// TIA Portal V20 export
FUNCTION "IF_Bool_Mapping" : Void   // FC104, SCL
// stored: SetENOAutomatically false
BEGIN
       // Des : I/O Interface signal Mapping //

   REGION BK

   REGION BK01

       "BK01"."X10-1 LEFT UNWINDER EXPEL BACKWARD" := "BA010AZCRBK01.00";
       "BK01"."X11-1 RIGHT UNWINDER EXPEL BACKWARD" := "BA010AZCRBK01.01";
       "BK01"."X12-1 UW SUPPORT UNIT TRANSFER BACKWARD" := "BA010AZCRBK01.02";
       "BK01"."X13-1 ELECTRODE SHAFT SUPPORTER DOWN" := "BA010AZCRBK01.03";
       "BK01"."X14-1 LEFT TENSION CHECK SENSOR" := "BA010AZCRBK01.04";
       "BK01"."X15-1 ELECTRODE FIX LEFT TOP PRESSURE SWITCH" := "BA010AZCRBK01.05";
     //"BK01"."X16-1 SPARE" := "BA010AZCRBK01.06";
     //"BK01"."X17-1 SPARE" := "BA010AZCRBK01.07";
       "BK01"."X10-2 LEFT UNWINDER EXPEL FORWARD" := "BA010AZCRBK01.10";
       "BK01"."X11-2 RIGHT UNWINDER EXPEL FORWARD" := "BA010AZCRBK01.11";
       "BK01"."X12-2 UW SUPPORT UNIT TRANSFER FORWARD" := "BA010AZCRBK01.12";
       "BK01"."X13-2 ELECTRODE SHAFT SUPPORTER UP" := "BA010AZCRBK01.13";
       "BK01"."X14-2 RIGHT TENSION CHECK SENSOR" := "BA010AZCRBK01.14";
       "BK01"."X15-2 ELECTRODE FIX LEFT BTM PRESSURE SWITCH" := "BA010AZCRBK01.15";
     //"BK01"."X16-2 SPARE" := "BA010AZCRBK01.14";
     //"BK01"."X17-2 SPARE" := "BA010AZCRBK01.15";

   END_REGION 

   REGION BK02

       "BK02"."X10-1 ELECTRODE FIX RIGHT TOP BACKWARD" := "BA010AZCRBK02.00";
       "BK02"."X10-2 ELECTRODE FIX RIGHT TOP FORWARD" := "BA010AZCRBK02.01";
       "BK02"."X12-1 ELECTRODE FIX RIGHT BTM BACKWARD" := "BA010AZCRBK02.02";
       "BK02"."X12-2 ELECTRODE FIX RIGHT BTM FORWARD" := "BA010AZCRBK02.03";
       "BK02"."X14-1 ELECTRODE FIX RIGHT TOP PRESSURE SWITCH" := "BA010AZCRBK02.04";
       "BK02"."X14-2 ELECTRODE FIX RIGHT BTM PRESSURE SWITCH" := "BA010AZCRBK02.05";
       "BK02"."X16-1 ELECTRODE CUTTER BACKWARD" := "BA010AZCRBK02.06";
       "BK02"."X16-2 ELECTRODE CUTTER FORWARD" := "BA010AZCRBK02.07";

   END_REGION

   REGION BK03
       "BK03"."X10-1 ELECTRODE FIX LEFT TOP BACKWARD" := "BA010AZCRBK03.00";
       "BK03"."X11-1 UNWINDER STOPPER BACKWARD" := "BA010AZCRBK03.01";
       "BK03"."X12-1 ELECTRODE FIX LEFT BTM BACKWARD" := "BA010AZCRBK03.02";
       //"BK03"."X13-1 DIGITAL PRESSURE SWITCH OUT1" := "BA010AZCRBK03.03";
       "BK03"."X14-1 ELECTRODE FIX LEFT TOP UP" := "BA010AZCRBK03.04";
       "BK03"."X15-1 FRAME COVER BACKWARD" := "BA010AZCRBK03.05";
       "BK03"."X16-1 ELECTRODE FIX LEFT BTM DOWN" := "BA010AZCRBK03.06";
     //"BK03"."X17-1 SPARE" := "BA010AZCRBK03.07";
       "BK03"."X10-2 ELECTRODE FIX LEFT TOP FORWARD" := "BA010AZCRBK03.10";
       "BK03"."X11-2 UNWINDER STOPPER FORWARD" := "BA010AZCRBK03.11";
       "BK03"."X12-2 ELECTRODE FIX LEFT BTM FORWARD" := "BA010AZCRBK03.12";
       //"BK03"."X13-2 DIGITAL PRESSURE SWITCH OUT2" := "BA010AZCRBK03.11";
       "BK03"."X14-2 ELECTRODE FIX LEFT TOP DOWN" := "BA010AZCRBK03.14";
       "BK03"."X15-2 FRAME COVER FORWARD" := "BA010AZCRBK03.15";
       "BK03"."X16-2 ELECTRODE FIX LEFT BTM UP" := "BA010AZCRBK03.16";
     //"BK03"."X17-2 SPARE":= "BA010AZCRBK03.15";

   END_REGION

   REGION BK04

       "BK04"."X10-1 SPLICING L-MODULE MOVER BACKWARD" := "BA010AZCRBK04.00";
       "BK04"."X11-1 SPLICING R-MODULE MOVER BACKWARD" := "BA010AZCRBK04.01";
       "BK04"."X12-1 ELECTRODE L-HOLDER MOVER FORWARD" := "BA010AZCRBK04.02";
       "BK04"."X13-1 ELECTRODE R-HOLDER MOVER FORWARD" := "BA010AZCRBK04.03";
       "BK04"."X14-1 TAPE LOADING TURN HOMING" := "BA010AZCRBK04.04";
       "BK04"."X15-1 TAPE ATTACH UNIT BACKWARD" := "BA010AZCRBK04.05";
       "BK04"."X16-1 TAPING VACUUM PRESSURE SWITCH" := "BA010AZCRBK04.06";
       //"BK04"."X17-1 SPARE" := "BA010AZCRBK04.07";
       "BK04"."X10-2 SPLICING L-MODULE MOVER FORWARD" := "BA010AZCRBK04.10";
       "BK04"."X11-2 SPLICING R-MODULE MOVER FORWARD" := "BA010AZCRBK04.11";
       "BK04"."X12-2 ELECTRODE L-HOLDER MOVER BACKWARD" := "BA010AZCRBK04.12";
       "BK04"."X13-2 ELECTRODE R-HOLDER MOVER BACKWARD" := "BA010AZCRBK04.13";
       "BK04"."X14-2 TAPE LOADING TURN ROTATE" := "BA010AZCRBK04.14";
       "BK04"."X15-2 TAPE ATTACH UNIT FORWARD" := "BA010AZCRBK04.15";
       //"BK04"."X16-2 SPARE":= "BA010AZCRBK04.14";
       //"BK04"."X17-2 SPARE":= "BA010AZCRBK04.15";

   END_REGION

   REGION bk05

       //"BK05"."X10-1 SPARE" := "BA010AZCRBK05.00";
       //"BK05"."X11-1 SPARE" := "BA010AZCRBK05.01";
       //"BK05"."X12-1 COMPENSATOR LIMIT SENSOR(-)" := "BA010AZCRBK05.02";
       //"BK05"."X13-1 COMPENSATOR LIMIT SENSOR(+)" := "BA010AZCRBK05.03";
       "BK05"."X14-1 FEEDER CYLINDER UP" := "BA010AZCRBK05.04";
       "BK05"."X15-1 VISION PUSHER SUPPORT UP" := "BA010AZCRBK05.05";
       "BK05"."X16-1 ELECTRODE NG BOX LOCK CYLINDER DOWN" := "BA010AZCRBK05.06";
       "BK05"."X17-1 UNWINDER DANCER SAFETY PIN IDLE POSITION" := "BA010AZCRBK05.07";
       //"BK05"."X10-2 SPARE":= "BA010AZCRBK05.08";
       //"BK05"."X11-2 SPARE":= "BA010AZCRBK05.09";
       //"BK05"."X12-2 COMPENSATOR HOMING SENSOR" := "BA010AZCRBK05.10";
       "BK05"."X13-2 COMPENSATOR SAFETY PIN IDLE POSITION" := "BA010AZCRBK05.13";
       "BK05"."X14-2 FEEDER CYLINDER DOWN" := "BA010AZCRBK05.14";
       "BK05"."X15-2 VISION PUSHER SUPPORT DOWN" := "BA010AZCRBK05.15";
       "BK05"."X16-2 ELECTRODE NG BOX LOCK CYLINDER UP" := "BA010AZCRBK05.16";
       //"BK05"."X17-2 SPARE":= "BA010AZCRBK05.15";

   END_REGION

   REGION bk06

       "BK06"."X10-1 NG & MANUAL INPUT CYLINDER UP" := "BA010AZCRBK06.00";
       "BK06"."X11-1 MAGAZINE LOCK CYLINDER DOWN":= "BA010AZCRBK06.01";
       "BK06"."X12-1 NG & MANUAL INPUT PAD VACUUM PRESSURE SWITCH":= "BA010AZCRBK06.02";
       //"BK06"."X13-1 NG & MANUAL INPUT LIMIT SENSOR(-)":= "BA010AZCRBK06.03";
       //"BK06"."X14-1 NG & MANUAL INPUT LIMIT SENSOR(+)":= "BA010AZCRBK06.04";
       //"BK06"."X15-1 NG & MANUAL INPUT MAGAZINE LIMIT SENSOR(-)":= "BA010AZCRBK06.05";
       //"BK06"."X16-1 NG & MANUAL INPUT MAGAZINE LIMIT SENSOR(+)":= "BA010AZCRBK06.06";
       "BK06"."X17-1 NG & MANUAL INPUT MAGAZINE ELECTRODE DETECTION SENSOR":= "BA010AZCRBK06.07";
       "BK06"."X10-2 NG & MANUAL INPUT CYLINDER DOWN":= "BA010AZCRBK06.10";
       "BK06"."X11-2 MAGAZINE LOCK CYLINDER UP":= "BA010AZCRBK06.11";
       //"BK06"."X12-2 NG & MANUAL INPUT VIBRATOR VACUUM PRESSURE SWITCH" := "BA010AZCRBK06.11";
       "BK06"."X13-2 NG & MANUAL INPUT HOMING SENSOR":= "BA010AZCRBK06.14";
       //"BK06"."X14-2 NG & MANUAL INPUT ELECTRODE DETECTION SENSOR":= "BA010AZCRBK06.13";
       //"BK06"."X15-2 NG & MANUAL INPUT MAGAZINE HOMING SENSOR":= "BA010AZCRBK06.14";
       //"BK06"."X16-2 SPARE":= "BA010AZCRBK06.14";
       "BK06"."X17-2 NG & MANUAL INPUT MAGAZINE DETECTION SENSOR":= "BA010AZCRBK06.17";

   END_REGION

   REGION bk07

       //"BK07"."X10-1 POSITION MOVING LIMIT SENSOR(-)" := "BA010AZCRBK07.00";
       //"BK07"."X11-1 POSITION MOVING LIMIT SENSOR(+)":= "BA010AZCRBK07.01";
       //"BK07"."X12-1 VISION HOMING SENSOR":= "BA010AZCRBK07.02";
       //"BK07"."X13-1 ELECTRODE NG KICKER HOMING SENSOR":= "BA010AZCRBK07.03";
       "BK07"."X14-1 ELECTRODE NG BOX FULL SENSOR":= "BA010AZCRBK07.04";
       "BK07"."X15-1 ELECTRODE NG BOX DETECT SENSOR":= "BA010AZCRBK07.05";
       "BK07"."X16-1 NG & MANUAL INPUT MAGAZINE FULL SENSOR":= "BA010AZCRBK07.06";
       //"BK07"."X17-1 MAGAZINE Z-AXIS SAFETY PIN POSITION SENSOR":= "BA010AZCRBK07.07";
       //"BK07"."X10-2 POSITION MOVING HOMING SENSOR":= "BA010AZCRBK07.08";
       //"BK07"."X11-2 CUTTER HOMING SENSOR":= "BA010AZCRBK07.09";
       //"BK07"."X12-2 SPARE":= "BA010AZCRBK07.10";
       //"BK07"."X13-2 ELECTRODE PASS KICKER HOMING SENSOR":= "BA010AZCRBK07.11";
       //"BK07"."X14-2 SPARE":= "BA010AZCRBK07.12";
       //"BK07"."X15-2 SPARE":= "BA010AZCRBK07.13";
       //"BK07"."X16-2 SPARE":= "BA010AZCRBK07.14";
       //"BK07"."X17-2 SPARE" := "BA010AZCRBK07.15";

   END_REGION

   REGION bk08

       "BK08"."X10-1 UW ELECTRODE FIX LEFT TOP V/C ON" := "BA010AZCRBK08.00";
       "BK08"."X10-2 UW ELECTRODE FIX LEFT TOP V/C OFF" := "BA010AZCRBK08.01";
       "BK08"."X12-1 UW ELECTRODE FIX LEFT BTM V/C ON" := "BA010AZCRBK08.02";
       "BK08"."X12-2 UW ELECTRODE FIX LEFT BTM V/C OFF" := "BA010AZCRBK08.03";
       "BK08"."X14-1 UW ELECTRODE FIX RIGHT TOP V/C ON" := "BA010AZCRBK08.04";
       "BK08"."X14-2 UW ELECTRODE FIX RIGHT TOP V/C OFF" := "BA010AZCRBK08.05";
       "BK08"."X16-1 UW ELECTRODE FIX RIGHT BTM V/C ON" := "BA010AZCRBK08.06";
       "BK08"."X16-2 UW ELECTRODE FIX RIGHT BTM V/C OFF" := "BA010AZCRBK08.07";

   END_REGION

   REGION bk09

       "BK09"."X10-1 NG & MANUAL INPUT VIBRATOR-1 ON" := "BA010AZCRBK09.00";
       "BK09"."X10-2 NG & MANUAL INPUT VIBRATOR-1 OFF" := "BA010AZCRBK09.01";
       "BK09"."X12-1 NG & MANUAL INPUT PAD VACUUM ON":= "BA010AZCRBK09.02";
       "BK09"."X12-2 NG & MANUAL INPUT PAD VACUUM OFF":= "BA010AZCRBK09.03";
       "BK09"."X14-1 NG & MANUAL INPUT VIBRATOR VACUUM ON" := "BA010AZCRBK09.04";
       "BK09"."X14-2 NG & MANUAL INPUT VIBRATOR VACUUM OFF":= "BA010AZCRBK09.05";
       "BK09"."X16-1 NG & MANUAL INPUT VIBRATOR-2 ON":= "BA010AZCRBK09.06";
       "BK09"."X16-2 NG & MANUAL INPUT VIBRATOR-2 OFF":= "BA010AZCRBK09.07";

   END_REGION

   REGION bk10

       "BK10"."X10-1 UW TAPE ATTACH V/C ON" := "BA010AZCRBK10.00";
       "BK10"."X10-2 UW TAPE ATTACH V/C OFF" := "BA010AZCRBK10.01";
       "BK10"."X12-1 CART DETECT CHECK LAMP" := "BA010AZCRBK10.02";
       //"BK10"."X12-2 SPARE" := "BA010AZCRBK10.03";
       //"BK10"."X14-1 SPARE" := "BA010AZCRBK10.04";
       //"BK10"."X14-2 SPARE" := "BA010AZCRBK10.05";
       //"BK10"."X16-1 SPARE" := "BA010AZCRBK10.06";
       //"BK10"."X16-2 SPARE" := "BA010AZCRBK10.07";
   END_REGION

   END_REGION

   REGION SBK

       REGION SBK01
           "SBK01"."X1-0 No EMG stop: Unwinder" := "BA010AZCRSBK01.00";
           "SBK01"."X2-1 No EMG stop: Reel cut" := "BA010AZCRSBK01.01";
           "SBK01"."X3-2 No EMG stop: Vision" := "BA010AZCRSBK01.02";
           "SBK01"."X4-3 No EMG stop: Conveyor" := "BA010AZCRSBK01.03";
           "SBK01"."X1-4 reserved" := "BA010AZCRSBK01.04";
           "SBK01"."X2-5 reserved" := "BA010AZCRSBK01.05";
           "SBK01"."X3-6 reserved" := "BA010AZCRSBK01.06";
           "SBK01"."X4-7 reserved" := "BA010AZCRSBK01.07";
           "SBK01"."X5-0 reserved" := "BA010AZCRSBK01.10";
           "SBK01"."X6-1 reserved" := "BA010AZCRSBK01.11";
           "SBK01"."X7-2 reserved" := "BA010AZCRSBK01.12";

       END_REGION

       REGION SBK02
           "SBK02"."X1-0 SCS box: SCS mode select, Setup" := "BA010AZCRSBK02.00";
           "SBK02"."X2-1 SCS box: SCS mode select, Disable" := "BA010AZCRSBK02.01";
           "SBK02"."X3-2 Frame Corver Detect Sensor" := "BA010AZCRSBK02.02";
           "SBK02"."X4-3  SAFETY DOOR LOCK7.INPUT" := "BA010AZCRSBK02.03";
           "SBK02"."X1-4 SCS box: SCS mode select, Auto" := "BA010AZCRSBK02.04";
           "SBK02"."X2-5 SPARE" := "BA010AZCRSBK02.05";
           "SBK02"."X3-6 SPARE" := "BA010AZCRSBK02.06";
           "SBK02"."X4-7 SAFETY DOOR LOCK7.INPUT" := "BA010AZCRSBK02.07";
           "SBK02"."X5-0 SCS box: Pendant required on, yellow" := "BA010AZCRSBK02.10";
           "SBK02"."X6-1 SCS box: SCS Disable mode selected, green" := "BA010AZCRSBK02.11";
           "SBK02"."X7-2 SAFETY DOOR LOCK7.OUTPUT" := "BA010AZCRSBK02.12";

       END_REGION

       REGION SBK03

           "SBK03"."X1-0 Roll change LH: Auto" := "BA010AZCRSBK03.00";
           "SBK03"."X2-1 Roll change RH: Auto" := "BA010AZCRSBK03.01";
           "SBK03"."X3-2 CART Detect Sensor 1" := "BA010AZCRSBK03.02";
           "SBK03"."X4-3 CART Detect Sensor 2" := "BA010AZCRSBK03.03";
           "SBK03"."X1-4 Roll change LH: Change" := "BA010AZCRSBK03.04";
           "SBK03"."X2-5 Roll change RH: Change" := "BA010AZCRSBK03.05";
           "SBK03"."X3-6 reserved" := "BA010AZCRSBK03.06";
           "SBK03"."X4-7 reserved" := "BA010AZCRSBK03.07";
           "SBK03"."X5-0 Roll change LH: Roll change in progress" := "BA010AZCRSBK03.10";
           "SBK03"."X6-1 Roll change RH: Roll change in progress" := "BA010AZCRSBK03.11";
           "SBK03"."X7-2 reserved" := "BA010AZCRSBK03.12";

       END_REGION


       REGION SBK04

           "SBK04"."X1-0 Gate EC TOP: Lock" := "BA010AZCRSBK04.00";
           "SBK04"."X2-1 Gate EC TOP: Reset" := "BA010AZCRSBK04.01";
           "SBK04"."X3-2 DIFFERENTIAL PRESSURE SWITCH 1 NC" := "BA010AZCRSBK04.02";
           "SBK04"."X4-3 DIFFERENTIAL PRESSURE SWITCH 2 NC" := "BA010AZCRSBK04.03";
           "SBK04"."X1-4 Gate EC TOP: Unlock" := "BA010AZCRSBK04.04";
           "SBK04"."X2-5 reserved" := "BA010AZCRSBK04.05";
           "SBK04"."X3-6 reserved" := "BA010AZCRSBK04.06";
           "SBK04"."X4-7 reserved" := "BA010AZCRSBK04.07";
           "SBK04"."X5-0 Gate EC TOP: Lock lamp on" := "BA010AZCRSBK04.10";
           "SBK04"."X6-1 Gate EC TOP: Unlock lamp on" := "BA010AZCRSBK04.11";
           "SBK04"."X7-2 Gate EC TOP: Reset lamp on" := "BA010AZCRSBK04.12";

       END_REGION

       REGION SBK05

           "SBK05"."X1-0 Gate EC LH: Lock" := "BA010AZCRSBK05.00";
           "SBK05"."X2-1 Gate EC LH: Reset" := "BA010AZCRSBK05.01";
           "SBK05"."X3-2 reserved" := "BA010AZCRSBK05.02";
           "SBK05"."X4-3 reserved" := "BA010AZCRSBK05.03";
           "SBK05"."X1-4 Gate EC LH: Unlock" := "BA010AZCRSBK05.04";
           "SBK05"."X2-5 reserved" := "BA010AZCRSBK05.05";
           "SBK05"."X3-6 reserved" := "BA010AZCRSBK05.06";
           "SBK05"."X4-7 reserved" := "BA010AZCRSBK05.07";
           "SBK05"."X5-0 Gate EC LH: Lock lamp on" := "BA010AZCRSBK05.10";
           "SBK05"."X6-1 Gate EC LH: Unlock lamp on" := "BA010AZCRSBK05.11";
           "SBK05"."X7-2 Gate EC LH: Reset lamp on" := "BA010AZCRSBK05.12";

       END_REGION

       REGION SBK06
           "SBK06"."X1-0 Gate EC.Top Close" := "BA010AZCRSBK06.00";
           "SBK06"."X2-1 Gate EC.LH Close" := "BA010AZCRSBK06.01";
           "SBK06"."X3-2 Gate EC.RH Close" := "BA010AZCRSBK06.02";
           "SBK06"."X4-3 reserved" := "BA010AZCRSBK06.03";
           "SBK06"."X1-4 Gate EC.Top Close" := "BA010AZCRSBK06.04";
           "SBK06"."X2-5 Gate EC.LH Close" := "BA010AZCRSBK06.05";
           "SBK06"."X3-6 Gate EC.RH Close" := "BA010AZCRSBK06.06";
           "SBK06"."X4-7 reserved" := "BA010AZCRSBK06.07";
           "SBK06"."X5-0 Gate EC.Top UnLock" := "BA010AZCRSBK06.10";
           "SBK06"."X6-1 Gate EC.LH UnLock" := "BA010AZCRSBK06.11";
           "SBK06"."X7-2 Gate EC.RH UnLock" := "BA010AZCRSBK06.12";

       END_REGION

       REGION SBK07
           "SBK07"."X1-0 Gate Cutter Close" := "BA010AZCRSBK07.00";
           "SBK07"."X2-1 Gate Magazine Close" := "BA010AZCRSBK07.01";
           "SBK07"."X3-2 Gate Conveyor Close" := "BA010AZCRSBK07.02";
           "SBK07"."X4-3 reserved" := "BA010AZCRSBK07.03";
           "SBK07"."X1-4 Gate Cutter Close" := "BA010AZCRSBK07.04";
           "SBK07"."X2-5 Gate Magazine Close" := "BA010AZCRSBK07.05";
           "SBK07"."X3-6 Gate Conveyor Close" := "BA010AZCRSBK07.06";
           "SBK07"."X4-7 reserved" := "BA010AZCRSBK07.07";
           "SBK07"."X5-0 Gate Cutter Unlock" := "BA010AZCRSBK07.10";
           "SBK07"."X6-1 Gate Magazine Unlock" := "BA010AZCRSBK07.11";
           "SBK07"."X7-2 Gate Conveyor Unlock" := "BA010AZCRSBK07.12";

       END_REGION

       REGION SBK08

           "SBK08"."X1-0 Gate EC RH: Lock" := "BA010AZCRSBK08.00";
           "SBK08"."X2-1 Gate EC RH: Reset" := "BA010AZCRSBK08.01";
           "SBK08"."X3-2 reserved" := "BA010AZCRSBK08.02";
           "SBK08"."X4-3 reserved" := "BA010AZCRSBK08.03";
           "SBK08"."X1-4 Gate EC RH: Unlock" := "BA010AZCRSBK08.04";
           "SBK08"."X2-5 reserved" := "BA010AZCRSBK08.05";
           "SBK08"."X3-6 reserved" := "BA010AZCRSBK08.06";
           "SBK08"."X4-7 reserved" := "BA010AZCRSBK08.07";
           "SBK08"."X5-0 Gate EC RH: Lock lamp on" := "BA010AZCRSBK08.10";
           "SBK08"."X6-1 Gate EC RH: Unlock lamp on" := "BA010AZCRSBK08.11";
           "SBK08"."X7-2 Gate EC RH: Reset lamp on" := "BA010AZCRSBK08.12";

       END_REGION

       REGION SBK09

           "SBK09"."X1-0 Gate ScrapBox: Lock" := "BA010AZCRSBK09.00";
           "SBK09"."X2-1 Gate ScrapBox : Reset" := "BA010AZCRSBK09.01";
           "SBK09"."X3-2 reserved" := "BA010AZCRSBK09.02";
           "SBK09"."X4-3 reserved" := "BA010AZCRSBK09.03";
           "SBK09"."X1-4 Gate ScrapBox : Unlock" := "BA010AZCRSBK09.04";
           "SBK09"."X2-5 reserved" := "BA010AZCRSBK09.05";
           "SBK09"."X3-6 reserved" := "BA010AZCRSBK09.06";
           "SBK09"."X4-7 reserved" := "BA010AZCRSBK09.07";
           "SBK09"."X5-0 Gate ScrapBox : Lock lamp on" := "BA010AZCRSBK09.10";
           "SBK09"."X6-1 Gate ScrapBox : Unlock lamp on" := "BA010AZCRSBK09.11";
           "SBK09"."X7-2 Gate ScrapBox : Reset lamp on" := "BA010AZCRSBK09.12";

       END_REGION

   END_REGION

   REGION PM
       REGION PM01

           "PM01"."AIRS01 UNWINDER LEFT AIR SHAFT ON" := "BA010AZCRPM01.00";
           //"PM01".SPARE := "BA010AZCRPM01.01";
           "PM01"."AIRS02 UNWINDER RIGHT AIR SHAFT ON" := "BA010AZCRPM01.02";
           //"PM01".SPARE_1:= "BA010AZCRPM01.03";
           //"PM01".SPARE_2 := "BA010AZCRPM05.00";
           //"PM01".SPARE_3 := "BA010AZCRPM05.01";
           //"PM01".SPARE_4 := "BA010AZCRPM06.00";
           //"PM01".SPARE_5 := "BA010AZCRPM06.01";
           "PM01"."C03 UNWINDER SUPPORT UNIT TRANSFER FORWARD" := "BA010AZCRPM01.10";
           "PM01"."C03 UNWINDER SUPPORT UNIT TRANSFER BACKWARD" := "BA010AZCRPM01.11";
           "PM01"."C04 ELECTRODE SHAFT SUPPORTER UP" := "BA010AZCRPM01.12";
           "PM01"."C04 ELECTRODE SHAFT SUPPORTER DOWN" := "BA010AZCRPM01.13";
           //"PM01".SPARE_2:= "BA010AZCRPM01.12";
           //"PM01".SPARE_3:= "BA010AZCRPM01.13";
           //"PM01".SPARE_4:= "BA010AZCRPM01.14";
           //"PM01".SPARE_5:= "BA010AZCRPM01.15";

       END_REGION

       REGION PM02

           "PM02"."C05 UNWINDER SPLICER RIGHT ELECTRODE FIX RIGHT TOP FORWARD" := "BA010AZCRPM02.00";
           "PM02"."C05 UNWINDER SPLICER RIGHT ELECTRODE FIX RIGHT TOP BACKWARD" := "BA010AZCRPM02.01";
           "PM02"."C06 UNWINDER SPLICER RIGHT ELECTRODE FIX RIGHT BTM FORWARD" := "BA010AZCRPM02.02";
           "PM02"."C06 UNWINDER SPLICER RIGHT ELECTRODE FIX RIGHT BTM BACKWARD" := "BA010AZCRPM02.03";
           "PM02"."C07 UNWINDER SPLICER RIGHT CUTTER FORWARD" := "BA010AZCRPM02.04";
           "PM02"."C07 UNWINDER SPLICER RIGHT CUTTER BACKWARD" := "BA010AZCRPM02.05";
           "PM02"."C08 UNWINDER SPLICER LEFT ELECTRODE FIX LEFT TOP FORWARD" := "BA010AZCRPM02.06";
           "PM02"."C08 UNWINDER SPLICER LEFT ELECTRODE FIX LEFT TOP BACKWARD" := "BA010AZCRPM02.07";
           "PM02"."C09 UNWINDER SPLICER LEFT ELECTRODE FIX LEFT BTM FORWARD" := "BA010AZCRPM02.10";
           "PM02"."C09 UNWINDER SPLICER LEFT ELECTRODE FIX LEFT BTM BACKWARD":= "BA010AZCRPM02.11";
           "PM02"."C10 UNWINDER SPLICER LEFT ELECTRODE FIX LEFT TOP DOWN":= "BA010AZCRPM02.12";
           "PM02"."C10 UNWINDER SPLICER LEFT ELECTRODE FIX LEFT TOP UP":= "BA010AZCRPM02.13";
           "PM02"."C11 UNWINDER SPLICER LEFT ELECTRODE FIX LEFT BTM UP":= "BA010AZCRPM02.14";
           "PM02"."C11 UNWINDER SPLICER LEFT ELECTRODE FIX LEFT BTM DOWN":= "BA010AZCRPM02.15";
           //"PM02".SPARE := "BA010AZCRPM02.14";
           //"PM02".SPARE_1:= "BA010AZCRPM02.15";

       END_REGION

       REGION PM03

           "PM03"."C12 UNWINDER SPLICER HOLDER SPLICING LEFT MODULE MOVER FORWARD" := "BA010AZCRPM03.00";
           "PM03"."C12 UNWINDER SPLICER HOLDER SPLICING LEFT MODULE MOVER BACKWARD":= "BA010AZCRPM03.01";
           "PM03"."C13 UNWINDER SPLICER HOLDER SPLICING RIGHT MODULE MOVER FORWARD":= "BA010AZCRPM03.02";
           "PM03"."C13 UNWINDER SPLICER HOLDER SPLICING RIGHT MODULE MOVER BACKWARD":= "BA010AZCRPM03.03";
           "PM03"."C14 UNWINDER SPLICER HOLDER ELECTRODE LEFT HOLDER MODULE MOVER FORWARD":= "BA010AZCRPM03.04";
           "PM03"."C14 UNWINDER SPLICER HOLDER ELECTRODE LEFT HOLDER MODULE MOVER BACKWARD":= "BA010AZCRPM03.05";
           "PM03"."C15 UNWINDER SPLICER HOLDER ELECTRODE RIGHT HOLDER MODULE MOVER FORWARD":= "BA010AZCRPM03.06";
           "PM03"."C15 UNWINDER SPLICER HOLDER ELECTRODE RIGHT HOLDER MODULE MOVER BACKWARD":= "BA010AZCRPM03.07";
           "PM03"."C16 UNWINDER SPLICER TAPE LOADING TURN ROTATE":= "BA010AZCRPM03.10";
           "PM03"."C16 UNWINDER SPLICER TAPE LOADING TURN HOME":= "BA010AZCRPM03.11";
           "PM03"."C17 UNWINDER SPLICER TAPE ATTACH UNIT FORWARD":= "BA010AZCRPM03.12";
           "PM03"."C17 UNWINDER SPLICER TAPE ATTACH UNIT BACKWARD":= "BA010AZCRPM03.13";
           //"PM03".SPARE:= "BA010AZCRPM03.12";
           //"PM03".SPARE_1:= "BA010AZCRPM03.13";
           //"PM03".SPARE_2:= "BA010AZCRPM03.14";
           //"PM03".SPARE_3:= "BA010AZCRPM03.15";

       END_REGION

       REGION PM04

           "PM04"."C18 UNWINDER STOPPER FORWARD" := "BA010AZCRPM04.00";
           "PM04"."C18 UNWINDER STOPPER BACKWARD":= "BA010AZCRPM04.01";
           "PM04"."C19 UNWINDER DANCER FORWARD":= "BA010AZCRPM04.02";
           "PM04"."C19 UNWINDER DANCER BACKWARD" := "BA010AZCRPM04.03";
           "PM04"."C20 FEEDER CYLINDER DOWN":= "BA010AZCRPM04.04";
           "PM04"."C20 FEEDER CYLINDER UP":= "BA010AZCRPM04.05";
           "PM04"."C21 NG & MANUAL INPUT CYLINDER DOWN":= "BA010AZCRPM04.06";
           "PM04"."C21 NG & MANUAL INPUT CYLINDER UP":= "BA010AZCRPM04.07";
           "PM04"."C22 MAGAZINE LOCK CYLINDER UP":= "BA010AZCRPM04.10";
           "PM04"."C22 MAGAZINE LOCK CYLINDER DOWN":= "BA010AZCRPM04.11";
           "PM04"."C23 VISION PUSHER SUPPORT DOWN":= "BA010AZCRPM04.12";
           "PM04"."C23 VISION PUSHER SUPPORT UP":= "BA010AZCRPM04.13";
           "PM04"."C24 ELECTRODE NG BOX LOCK CYLINDER UP" := "BA010AZCRPM04.14";
           "PM04"."C24 ELECTRODE NG BOX LOCK CYLINDER DOWN":= "BA010AZCRPM04.15";
           "PM04"."C25 FRAME COVER FORWARD":= "BA010AZCRPM04.16";
           "PM04"."C25 FRAME COVER BACKWARD":= "BA010AZCRPM04.17";

       END_REGION

       REGION PM05

           "PM05"."c1 LEFT UNWINDER EXPEL FORWARD" := "BA010AZCRPM05.00";
           "PM05"."c1 LEFT UNWINDER EXPEL BACKWARD" := "BA010AZCRPM05.01";
           //"PM05".SPARE_1 := "BA010AZCRPM05.02";
           //"PM05".SPARE_2 := "BA010AZCRPM05.03";
           //"PM05".SPARE_3 := "BA010AZCRPM05.04";
           //"PM05".SPARE_4 := "BA010AZCRPM05.05";
           //"PM05".SPARE_5 := "BA010AZCRPM05.06";
           //"PM05".SPARE_6 := "BA010AZCRPM05.07";
           //"PM05".SPARE_7 := "BA010AZCRPM05.08";
           //"PM05".SPARE_8 := "BA010AZCRPM05.09";
           //"PM05".SPARE_9 := "BA010AZCRPM05.10";
           //"PM05".SPARE_10 := "BA010AZCRPM05.11";
           //"PM05".SPARE_11 := "BA010AZCRPM05.12";
           //"PM05".SPARE_12 := "BA010AZCRPM05.13";
           //"PM05".SPARE_13 := "BA010AZCRPM05.14";
           //"PM05".SPARE_14 := "BA010AZCRPM05.15";

       END_REGION

       REGION PM06

           "PM06"."c2 RIGHT UNWINDER EXPEL FORWARD" := "BA010AZCRPM06.00";
           "PM06"."c2 RIGHT UNWINDER EXPEL BACKWARD" := "BA010AZCRPM06.01";
           //"PM06".SPARE_1 := "BA010AZCRPM06.02";
           //"PM06".SPARE_2 := "BA010AZCRPM06.03";
           //"PM06".SPARE_3 := "BA010AZCRPM06.04";
           //"PM06".SPARE_4 := "BA010AZCRPM06.05";
           //"PM06".SPARE_5 := "BA010AZCRPM06.06";
           //"PM06".SPARE_6 := "BA010AZCRPM06.07";
           //"PM06".SPARE_7 := "BA010AZCRPM06.08";
           //"PM06".SPARE_8 := "BA010AZCRPM06.09";
           //"PM06".SPARE_9 := "BA010AZCRPM06.10";
           //"PM06".SPARE_10 := "BA010AZCRPM06.11";
           //"PM06".SPARE_11 := "BA010AZCRPM06.12";
           //"PM06".SPARE_12 := "BA010AZCRPM06.13";
           //"PM06".SPARE_13 := "BA010AZCRPM06.14";
           //"PM06".SPARE_14 := "BA010AZCRPM06.15";

       END_REGION

   END_REGION

   REGION ET200SP

       REGION ET200SP JBOX
           REGION SP501

               "ET500SP_501"."SP501.00 CONTROL DC POWER TRIPPED E156CB" := "BA010AZCRSP501.00";
               "ET500SP_501"."SP501.01 SAFETY DC POWER TRIPPED E218CB" := "BA010AZCRSP501.01";
               //"ET500SP_501".SPARE1 := "BA010AZCRSP501.02";
               //"ET500SP_501".SPARE2 := "BA010AZCRSP501.03";
               "ET500SP_501"."SP501.04 Vision STO" := "BA010AZCRSP501.04";
               "ET500SP_501"."SP501.05 Vision Judgment" := "BA010AZCRSP501.05";
               //"ET500SP_501".SPARE3 := "BA010AZCRSP501.07";
               //"ET500SP_501".SPARE4 := "BA010AZCRSP501.08";
               //"ET500SP_501".SPARE5 := "BA010AZCRSP501.09";
               //"ET500SP_501".SPARE6 := "BA010AZCRSP501.10";
               //"ET500SP_501".SPARE7 := "BA010AZCRSP501.11";
               //"ET500SP_501".SPARE8 := "BA010AZCRSP501.12";
               //"ET500SP_501".SPARE9 := "BA010AZCRSP501.13";
               //"ET500SP_501".SPARE10 := "BA010AZCRSP501.14";
               //"ET500SP_501".SPARE11 := "BA010AZCRSP501.15";
               //"ET500SP_501".SPARE12 := "BA010AZCRSP501.16";

           END_REGION

           REGION SP502

               //"ET500SP_502".SPARE1 := "BA010AZCRSP502.00";
               //"ET500SP_502".SPARE2 := "BA010AZCRSP502.01";
               //"ET500SP_502".SPARE3 := "BA010AZCRSP502.02";
               //"ET500SP_502".SPARE4 := "BA010AZCRSP502.03";
               //"ET500SP_502".SPARE5 := "BA010AZCRSP502.04";
               //"ET500SP_502".SPARE6 := "BA010AZCRSP502.05";
               //"ET500SP_502".SPARE7 := "BA010AZCRSP502.06";
               //"ET500SP_502".SPARE8 := "BA010AZCRSP502.07";
               //"ET500SP_502".SPARE9 := "BA010AZCRSP502.08";
               //"ET500SP_502".SPARE10 := "BA010AZCRSP502.09";
               //"ET500SP_502".SPARE11 := "BA010AZCRSP502.10";
               //"ET500SP_502".SPARE12 := "BA010AZCRSP502.11";
               //"ET500SP_502".SPARE13 := "BA010AZCRSP502.12";
               //"ET500SP_502".SPARE14 := "BA010AZCRSP502.13";
               //"ET500SP_502".SPARE15 := "BA010AZCRSP502.14";
               //"ET500SP_502".SPARE16 := "BA010AZCRSP502.15";

           END_REGION

           REGION SP503

               "ET500SP_503"."SP503.00 LEFT UNWINDER RADIUS MEASURE" :="BA010AZCRSP503.00";
               "ET500SP_503"."SP503.01 RIGHT UNWINDER RADIUS MEASURE":="BA010AZCRSP503.01";
               "ET500SP_503"."SP503.02 UNWINDER LOADCELL":="BA010AZCRSP503.02";
               "ET500SP_503"."SP503.03 CUTTER EPC SENSOR" := "BA010AZCRSP503.03";

           END_REGION

           REGION SP504

               "ET500SP_504"."SP504.00 UNWINDER DANCER ENCODER" := "BA010AZCRSP504.00";
               //"ET500SP_504".SPARE1 := "BA010AZCRSP504.01";
               //"ET500SP_504".SPARE2 := "BA010AZCRSP504.02";
               //"ET500SP_504".SPARE3 := "BA010AZCRSP504.03";

           END_REGION
           REGION SP505

               "ET500SP_505"."SP505.00 UNWINDER DANCER ELECTRO-PNEUMATIC REGULATOR" := "BA010AZCRSP505.00";
               //"ET500SP_505".SPARE1 := "BA010AZCRSP505.01";
               //"ET500SP_505".SPARE2 := "BA010AZCRSP505.02";
               //"ET500SP_505".SPARE3 := "BA010AZCRSP505.03";

           END_REGION
           REGION SP506
               //"ET500SP_506"."SP506.00 Tab Sensor" := "MeasuringInput_FeedingRollAxisB_Tab_Interface_Address";
               //"ET500SP_506"."SP506.01 Tape Sensor" := "MeasuringInput_FeedingRollAxisB_Tape_Interface_Address";
               "ET500SP_506"."SP506.02 VISION TRIGGER SENSOR" := "BA010AZCRSP506.02";
               "ET500SP_506"."SP506.03 ELECTRODE PASS KICKER DETECT SENSOR" := "BA010AZCRSP506.03";
               //"ET500SP_506"."SP506.04 OutputCam_FeedingRollAxisB" := "BA010AZCRSP506.04";
               //"ET500SP_506"."SP506.05 OutputCam_ElectrodCutterAxisZ" := "BA010AZCRSP506.05";
               "ET500SP_506"."SP506.06 VISION CONTROLLER TRIGGER" := "BA010AZCRSP506.06";
               //"ET500SP_506"."SP506.07 OutputCam_NgKickerAxisZ" := "BA010AZCRSP506.07";
               //"ET500SP_506".SPARE1 := "BA010AZCRSP506.08";

           END_REGION
           REGION SP507

               "ET500SP_507"."SP507.00 ELECTRODE NG KICKER DETECT SENSOR" := "BA010AZCRSP507.00";
               "ET500SP_507"."SP507.01 ELECTRODE DETECT COLOR SENSOR #1" := "BA010AZCRSP507.01";
               "ET500SP_507"."SP507.02 ELECTRODE DETECT COLOR SENSOR #2" := "BA010AZCRSP507.02";
               //"ET500SP_507".SPARE1 := "BA010AZCRSP507.03";
               //"ET500SP_507"."SP507.04 OutputCam_PassKickerAxisZ" := "BA010AZCRSP507.04";
               //"ET500SP_507".SPARE2 := "BA010AZCRSP507.05";
               //"ET500SP_507".SPARE3 := "BA010AZCRSP507.06";
               //"ET500SP_507".SPARE4 := "BA010AZCRSP507.07";
               //"ET500SP_507".SPARE5 := "BA010AZCRSP507.08";

           END_REGION
           REGION SP508

               "ET500SP_508"."SP508.00 PHMI-1 EMERGENCY STOP" := "BA010AZCRSP508.00";
               "ET500SP_508"."SP508.01 PHMI-1 ENABLE SWITCH" := "BA010AZCRSP508.01";
               "ET500SP_508"."SP508.02 PHMI-2 EMERGENCY STOP" := "BA010AZCRSP508.02";
               "ET500SP_508"."SP508.03 PHMI-2 ENABLE SWITCH" := "BA010AZCRSP508.03";
               //"ET500SP_508".SPARE1 := "BA010AZCRSP508.04";
               //"ET500SP_508".SPARE2 := "BA010AZCRSP508.05";
               //"ET500SP_508".SPARE3 := "BA010AZCRSP508.06";
               //"ET500SP_508".SPARE4 := "BA010AZCRSP508.07";

           END_REGION
           REGION 509

               "ET500SP_509"."SP509.00 UNWINDER EPCC01 INTERKOCK" := "BA010AZCRSP509.00";
               "ET500SP_509"."SP509.01 UNWINDER EPCC02 INTERLOCK" := "BA010AZCRSP509.01";
               "ET500SP_509"."SP509.02 UNWINDER EPCC03 INTERLOCK" := "BA010AZCRSP509.02";
               //"ET500SP_509".SPARE1 := "BA010AZCRSP509.03";
               //"ET500SP_509".SPARE2 := "BA010AZCRSP509.04";
               //"ET500SP_509".SPARE3 := "BA010AZCRSP509.05";
               //"ET500SP_509".SPARE4 := "BA010AZCRSP509.06";
               //"ET500SP_509".SPARE5 := "BA010AZCRSP509.07";

           END_REGION
           REGION SP510

           END_REGION
           REGION SP511

           END_REGION
           REGION SP512

           END_REGION
           REGION SP513

               "ET500SP_513"."SP513.00 LEFT UNWINDER RADIUS SENSOR" := "BA010AZCRSP513.00";
               "ET500SP_513"."SP513.01 RIGHT UNWINDER RADIUS SENSOR" := "BA010AZCRSP513.01";
               //"ET500SP_513".SPARE1 := "BA010AZCRSP513.02";
               //"ET500SP_513".SPARE2 := "BA010AZCRSP513.03";

           END_REGION
       END_REGION

       REGION ET200SP D1Panel
           REGION SP201

               "ET200SP_201"."SP201.00 AUTO INITIATE PBL (GREEN)" :="BA010AZCRSP201.00";
               "ET200SP_201"."SP201.01 STOP PBL (RED)" := "BA010AZCRSP201.01";
               //"ET200SP_201".SPARE1 := "BA010AZCRSP201.02";
               //"ET200SP_201".SPARE2 := "BA010AZCRSP201.03";
               //"ET200SP_201".SPARE3 := "BA010AZCRSP201.04";
               //"ET200SP_201".SPARE4 := "BA010AZCRSP201.05";
               //"ET200SP_201".SPARE5 := "BA010AZCRSP201.06";
               //"ET200SP_201".SPARE6 := "BA010AZCRSP201.07";
               "ET200SP_201"."SP201.08 MAIN HMI POWER TRIPPED E110CB" := "BA010AZCRSP201.10";
               //"ET200SP_201".SPARE7 := "BA010AZCRSP201.09";
               //"ET200SP_201".SPARE8 := "BA010AZCRSP201.10";
               //"ET200SP_201".SPARE9 := "BA010AZCRSP201.11";
               //"ET200SP_201".SPARE10 := "BA010AZCRSP201.12";
               //"ET200SP_201".SPARE11 := "BA010AZCRSP201.13";
               //"ET200SP_201".SPARE12 := "BA010AZCRSP201.14";
               //"ET200SP_201".SPARE13 := "BA010AZCRSP201.15";

           END_REGION
           REGION SP202

               "ET200SP_202"."SP202.00 AUTO INITIATE PBL LAMP ON (GREEN)" := "BA010AZCRSP202.00";
               "ET200SP_202"."SP202.01 STOP PBL LAMP ON (RED)" := "BA010AZCRSP202.01";
               //"ET200SP_202".SPARE1 := "BA010AZCRSP202.02";
               "ET200SP_202"."SP202.03 ENABLE PBL LAMP ON (BLACK)" := "BA010AZCRSP202.03";
               "ET200SP_202"."SP202.04 SAFETY RESET PBL LAMP ON (BLUE)" := "BA010AZCRSP202.04";
               //"ET200SP_202".SPARE2 := "BA010AZCRSP202.05";
               //"ET200SP_202".SPARE3 := "BA010AZCRSP202.06";
               //"ET200SP_202".SPARE4 := "BA010AZCRSP202.07";
               "ET200SP_202"."SP202.08 TOWER LAMP 1 ON (RED)" := "BA010AZCRSP202.10";
               "ET200SP_202"."SP202.09 TOWER LAMP 2 ON (AMBER)" := "BA010AZCRSP202.11";
               "ET200SP_202"."SP202.10 TOWER LAMP 3 ON (GREEN)" := "BA010AZCRSP202.12";
               "ET200SP_202"."SP202.11 TOWER LAMP 4 ON (WHITE)" := "BA010AZCRSP202.13";
               "ET200SP_202"."SP202.12 TOWER LAMP 5 ON (BLUE)" := "BA010AZCRSP202.14";
               "ET200SP_202"."SP202.13 TOWER LAMP 6 ON (BUZZER)" := "BA010AZCRSP202.15";
               //"ET200SP_202".SPARE5 := "BA010AZCRSP202.14";
               //"ET200SP_202".SPARE6 := "BA010AZCRSP202.15";

           END_REGION
           REGION SP203

               "ET200SP_203"."SP203.00 Main OP: mode select, Auto" := "BA010AZCRSP203.00";
               "ET200SP_203"."SP203.01 Main OP: home (GREEN)" := "BA010AZCRSP203.01";
               "ET200SP_203"."SP203.02 Main OP: safety reset (BLUE)" := "BA010AZCRSP203.02";
               "ET200SP_203"."SP203.03 Main OP: SCS mode select, Auto" := "BA010AZCRSP203.03";
               "ET200SP_203"."SP203.04 Main OP: mode select, Manual" := "BA010AZCRSP203.04";
               "ET200SP_203"."SP203.05 Main OP: enable" := "BA010AZCRSP203.05";
               "ET200SP_203"."SP203.06 Main OP: SCS mode select, Setup" := "BA010AZCRSP203.06";
               "ET200SP_203"."SP203.07 Main OP: SCS mode select, Disable" := "BA010AZCRSP203.07";

           END_REGION
           REGION SP204

               "ET200SP_204"."SP204.00 Main OP: Emergency stop" := "BA010AZCRSP204.00";
               //"ET200SP_204".SPARE1 := "BA010AZCRSP204.01";
               //"ET200SP_204".SPARE2 := "BA010AZCRSP204.02";
               //"ET200SP_204".SPARE3 := "BA010AZCRSP204.03";
               "ET200SP_204".RESERVED := "BA010AZCRSP204.04";
               //"ET200SP_204".SPARE4 := "BA010AZCRSP204.05";
               //"ET200SP_204".SPARE5 := "BA010AZCRSP204.06";
               //"ET200SP_204".SPARE6 := "BA010AZCRSP204.07";

           END_REGION
           REGION SP205

               "ET200SP_205"."SP205.00 Main OP: pendant required on, yellow" := "BA010AZCRSP205.00";
               //"ET200SP_205".SPARE1 := "BA010AZCRSP205.01";
               "ET200SP_205"."SP205.02 Main OP: home on, green" := "BA010AZCRSP205.02";
               //"ET200SP_205".SPARE2 := "BA010AZCRSP205.03";
               //"ET200SP_205".SPARE3 := "BA010AZCRSP205.04";
               //"ET200SP_205".SPARE4 := "BA010AZCRSP205.05";
               //"ET200SP_205".SPARE5 := "BA010AZCRSP205.06";
               "ET200SP_205"."SP205.07 Main OP: SCS Disable mode selected, green" := "BA010AZCRSP205.07";

           END_REGION
       END_REGION


   END_REGION

   REGION PLC CPU

       REGION DI1

           "DI1"."MOTOR POWER TRIPPED E202CB" := "BA010AZCRMP101.00";
           "DI1"."REELCUT CONVEYOR RING BLOW POWER TRIPPED" := "BA010AZCRMP101.01";
           "DI1"."STACKING-1 CONVEYOR RING BLOW POWER TRIPPED E214CB" := "BA010AZCRMP101.02";
           "DI1"."STACKING-2 CONVEYOR RING BLOW POWER TRIPPED E220CB" := "BA010AZCRMP101.03";
           //"DI1"."SPARE1" := "BA010AZCRDI1.04";
           "DI1"."E6404PWS CONTROLLER POWER SMPS AC POWER TRIPPED E320CB" := "BA010AZCRMP101.05";
           "DI1"."E6704PWS CONTROLLER POWER SMPS AC POWER TRIPPED E326CB" := "BA010AZCRMP101.06";
           "DI1"."E6804PWS SAFETY POWER SMPS AC POWER TRIPPED E332CB" := "BA010AZCRMP101.07";
           //"DI1"."SPARE2" := "BA010AZCRDI1.08";
           "DI1"."POWER METER POWER TRIPPED E720CB" := "BA010AZCRMP101.11";
           "DI1"."POWER METER CONTROL POWER TRIPPED E726CB" := "BA010AZCRMP101.12";
           //"DI1"."SPARE3" := "BA010AZCRDI1.11";
           "DI1"."PROCESSOR POWER ON TRIPPED E4116CB" := "BA010AZCRMP101.14";
           "DI1"."PROGRAMMING POWER OUTLET TRIPPED E4156CB" := "BA010AZCRMP101.15";
           //"DI1"."SPARE4" := "BA010AZCRDI1.14";
           "DI1"."PANEL LED POWER TRIPPED E4304CB" := "BA010AZCRMP101.17";
           //"DI1"."SPARE5" := "BA010AZCRDI1.16";
           "DI1"."PLC POWER SMPS DC OK E4404PWS" := "BA010AZCRMP101.21";
           "DI1"."CONTROL LEVEL HUB POWER TRIPPED E4420CB" := "BA010AZCRMP101.22";
           "DI1"."MAIN HMI POWER TRIPPED E4426CB" := "BA010AZCRMP101.23";
           "DI1"."PORTABLE HMI POWER TRIPPED E4432CB" := "BA010AZCRMP101.24";
           "DI1"."PORTABLE HMI POWER TRIPPED E4456CB" := "BA010AZCRMP101.25";
           //"DI1"."SPARE6" := "BA010AZCRDI1.22";
           //"DI1"."SPARE7" := "BA010AZCRDI1.23";
           "DI1"."120VAC CONTROL POWER TR PRIMARY TRIPPED E5100CB" := "BA010AZCRMP101.30";
           "DI1"."120VAC CONTROL POWER TR SECONDARY TRIPPED E5110CB" := "BA010AZCRMP101.31";
           "DI1"."CONTROL POWER ON TRIPPED E5116CB" := "BA010AZCRMP101.32";
           "DI1"."VISION MONITOR POWER STRIP OUTLET POWER TRIPPED E5160CB" := "BA010AZCRMP101.33";
           "DI1"."MCU & RFD HANDY POWER STRIP OUTLET POWER TRIPPED E5166CB" := "BA010AZCRMP101.34";
           "DI1"."VISION LIGHT CONTROLLER POWER STRIP OUTLET POWER TRIPPED E5172CB" := "BA010AZCRMP101.35";
           //"DI1"."SPARE8" := "BA010AZCRDI1.30";
           "DI1"."FFU POWER-1 POWER TRIPPED E3222CB" := "BA010AZCRMP101.37";


       END_REGION

       REGION DI2

           //"DI2"."SPARE1" := "BA010AZCRDI2.00";
           "DI2"."CONTROL POWER SMPS DC OK E6104PWS" := "BA010AZCRMP102.01";
           "DI2"."ET200MP I/O OUTPUT POWER TRIPPED E6154CB" := "BA010AZCRMP102.02";
           "DI2"."JUNCTION BOX CONTROL POWER TRIPPED E6180CB" := "BA010AZCRMP102.03";
           "DI2"."CLASS 2 SMPS POWER TRIPPED E6204CB" := "BA010AZCRMP102.04";
           "DI2"."CLASS 2 SMPS MONITORING E6206PWS" := "BA010AZCRMP102.05";
           "DI2"."ET200ECO PN-1 POWER TRIPPED E6220CB" := "BA010AZCRMP102.06";
           "DI2"."ET200ECO PN-2 POWER TRIPPED E6224CB" := "BA010AZCRMP102.07";
           "DI2"."ET200ECO PN-3 POWER TRIPPED E6228CB" := "BA010AZCRMP102.10";
           //"DI2"."SPARE2" := "BA010AZCRDI2.09";
           "DI2"."PANEL FAN POWER TRIPPED E6304CB" := "BA010AZCRMP102.12";
           //"DI2"."SPARE3" := "BA010AZCRDI2.11";
           "DI2"."CONTROLLER POWER SMPS DC OK E6404PWS" := "BA010AZCRMP102.14";
           "DI2"."CONTROLLER DC POWER TRIPPED E6406CB" := "BA010AZCRMP102.15";
           "DI2"."SERVO CONTROL POWER TRIPPED E6416CB" := "BA010AZCRMP102.16";
           "DI2"."MANIFOLD-1 CONTROL POWER TRIPPED E6422CB" := "BA010AZCRMP102.17";
           //"DI2"."SPARE4" := "BA010AZCRDI2.16";
           "DI2"."RFID POWER TRIPPED E6456CB" := "BA010AZCRMP102.21";
           "DI2"."QR READER POWER TRIPPED E6462CB" := "BA010AZCRMP102.22";
           "DI2"."QR READER POWER TRIPPED E6468CB" := "BA010AZCRMP102.23";
           //"DI2"."SPARE5" := "BA010AZCRDI2.20";
           //"DI2"."SPARE6" := "BA010AZCRDI2.21";
           "DI2"."CONTROLLER POWER SMPS DC OK E6704PWS" := "BA010AZCRMP102.26";
           "DI2"."CONTROLLER DC POWER TRIPPED E6706CB" := "BA010AZCRMP102.27";
           "DI2"."HANDY QR READER POWER TRIPPED E6716CB" := "BA010AZCRMP102.30";
           "DI2"."VISION CONTROLLER POWER TRIPPED E6722CB" := "BA010AZCRMP102.31";
           "DI2"."LINE LASER MODULE-1 POWER TRIPPED E6728CB" := "BA010AZCRMP102.32";
           "DI2"."LINE LASER MODULE-2 POWER TRIPPED E6734CB" := "BA010AZCRMP102.33";
           "DI2"."EPC CONTROLLER-1 POWER TRIPPED E6756CB" := "BA010AZCRMP102.34";
           "DI2"."EPC CONTROLLER-2 POWER TRIPPED E6762CB" := "BA010AZCRMP102.35";
           "DI2"."EPC CONTROLLER-3 POWER TRIPPED E6768CB" := "BA010AZCRMP102.36";
           "DI2"."DRIVE-CLIQ HUB POWER TRIPPED E6774CB" := "BA010AZCRMP102.37";


       END_REGION

       REGION DI3

           "DI3"."EQUIPMENT LED POWER TRIPPED E6780CB" := "BA010AZCRMP103.00";
           "DI3"."MOTOR POWER MC COIL POWER TRIPPED E6786CB" := "BA010AZCRMP103.01";
           "DI3"."SAFETY POWER SMPS DC OK E6804PWS" := "BA010AZCRMP103.02";
           "DI3"."SAFETY DC POWER TRIPPED E6808CB" := "BA010AZCRMP103.03";
           "DI3"."ET200SP I/O SAFETY POWER TRIPPED E6816CB" := "BA010AZCRMP103.04";
           "DI3"."JUNCTION BOX CONTROL POWER TRIPPED E6836CB" := "BA010AZCRMP103.05";
           "DI3"."ET200ECO PN-SAFETY-1 POWER TRIPPED E6856CB" := "BA010AZCRMP103.06";
           //"DI3"."SPARE1" := "BA010AZCRDI3.07";
           //"DI3"."SPARE2" := "BA010AZCRDI3.08";
           //"DI3"."SPARE3" := "BA010AZCRDI3.09";
           //"DI3"."SPARE4" := "BA010AZCRDI3.10";
           //"DI3"."SPARE5" := "BA010AZCRDI3.11";
           //"DI3"."SPARE6" := "BA010AZCRDI3.12";
           //"DI3"."SPARE7" := "BA010AZCRDI3.13";
           //"DI3"."SPARE8" := "BA010AZCRDI3.14";
           //"DI3"."SPARE9" := "BA010AZCRDI3.15";
           //"DI3"."SPARE10" := "BA010AZCRDI3.16";
           //"DI3"."SPARE11" := "BA010AZCRDI3.17";
           //"DI3"."SPARE12" := "BA010AZCRDI3.18";
           //"DI3"."SPARE13" := "BA010AZCRDI3.19";
           //"DI3"."SPARE14" := "BA010AZCRDI3.20";
           //"DI3"."SPARE15" := "BA010AZCRDI3.21";
           //"DI3"."SPARE16" := "BA010AZCRDI3.22";
           //"DI3"."SPARE17" := "BA010AZCRDI3.23";
           //"DI3"."SPARE18" := "BA010AZCRDI3.24";
           //"DI3"."SPARE19" := "BA010AZCRDI3.25";
           //"DI3"."SPARE20" := "BA010AZCRDI3.26";
           //"DI3"."SPARE21" := "BA010AZCRDI3.27";
           //"DI3"."SPARE22" := "BA010AZCRDI3.28";
           //"DI3"."SPARE23" := "BA010AZCRDI3.29";
           //"DI3"."SPARE24" := "BA010AZCRDI3.30";
           //"DI3"."SPARE25" := "BA010AZCRDI3.31";


       END_REGION

       REGION DQ1

           "DQ1"."EQUIPMENT LED LAMP RELAY ON" := "BA010AZCRMP104.00";
           //"DQ1"."SPARE1" := "BA010AZCRDQ1.01";
           //"DQ1"."SPARE2" := "BA010AZCRDQ1.02";
           "DQ1"."CLASS2 SMPS ALARM RESET" := "BA010AZCRMP104.03";
           //"DQ1"."SPARE3" := "BA010AZCRDQ1.04";
           //"DQ1"."SPARE4" := "BA010AZCRDQ1.05";
           //"DQ1"."SPARE5" := "BA010AZCRDQ1.06";
           //"DQ1"."SPARE6" := "BA010AZCRDQ1.07";
           //"DQ1"."SPARE7" := "BA010AZCRDQ1.08";
           //"DQ1"."SPARE8" := "BA010AZCRDQ1.09";
           //"DQ1"."SPARE9" := "BA010AZCRDQ1.10";
           //"DQ1"."SPARE10" := "BA010AZCRDQ1.11";
           //"DQ1"."SPARE11" := "BA010AZCRDQ1.12";
           //"DQ1"."SPARE12" := "BA010AZCRDQ1.13";
           //"DQ1"."SPARE13" := "BA010AZCRDQ1.14";
           //"DQ1"."SPARE14" := "BA010AZCRDQ1.15";
           //"DQ1"."SPARE15" := "BA010AZCRDQ1.16";
           //"DQ1"."SPARE16" := "BA010AZCRDQ1.17";
           //"DQ1"."SPARE17" := "BA010AZCRDQ1.18";
           //"DQ1"."SPARE18" := "BA010AZCRDQ1.19";
           //"DQ1"."SPARE19" := "BA010AZCRDQ1.20";
           //"DQ1"."SPARE20" := "BA010AZCRDQ1.21";
           //"DQ1"."SPARE21" := "BA010AZCRDQ1.22";
           //"DQ1"."SPARE22" := "BA010AZCRDQ1.23";
           //"DQ1"."SPARE23" := "BA010AZCRDQ1.24";
           //"DQ1"."SPARE24" := "BA010AZCRDQ1.25";
           //"DQ1"."SPARE25" := "BA010AZCRDQ1.26";
           //"DQ1"."SPARE26" := "BA010AZCRDQ1.27";
           //"DQ1"."SPARE27" := "BA010AZCRDQ1.28";
           //"DQ1"."SPARE28" := "BA010AZCRDQ1.29";
           //"DQ1"."SPARE29" := "BA010AZCRDQ1.30";
           //"DQ1"."SPARE30" := "BA010AZCRDQ1.31";


       END_REGION

       REGION FDI1

           "FDI1"."MANIFOLD-1 SOL POWER MC FEEDBACK" := "BA010AZCRMP105.00";
           "FDI1"."MANIFOLD-2 SOL POWER MC FEEDBACK" := "BA010AZCRMP105.01";
           //"FDI1"."SPARE1" := "BA010AZCRFDI1.02";
           //"FDI1"."SPARE2" := "BA010AZCRFDI1.03";
           "FDI1"."FFU POWER MC 1 FEEDBACK" := "BA010AZCRMP105.04";
           "FDI1"."FFU POWER MC 2 FEEDBACK" := "BA010AZCRMP105.05";
           //"FDI1"."SPARE3" := "BA010AZCRFDI1.06";
           //"FDI1"."SPARE4" := "BA010AZCRFDI1.07";


       END_REGION

       REGION FDQ1

           "FDQ1"."MANIFOLD-1 SOL POWER MC ON" := "BA010AZCRMP106.00";
           //"FDQ1"."SPARE1" := "BA010AZCRFDQ1.01";
           //"FDQ1"."SPARE2" := "BA010AZCRFDQ1.02";
           //"FDQ1"."SPARE3" := "BA010AZCRFDQ1.03";
           "FDQ1"."FFU POWER MC ON 1" := "BA010AZCRMP106.04";
           "FDQ1"."FFU POWER MC ON 2" := "BA010AZCRMP106.05";
           //"FDQ1"."SPARE4" := "BA010AZCRFDQ1.06";
           //"FDQ1"."SPARE5" := "BA010AZCRFDQ1.07";


       END_REGION


   END_REGION
END_FUNCTION
